(* IEC 61131-3 sources: teller/JD_Teller_LC2_V11/Class/Box_Editor_Preview_TC, 1 file *)

(* ---- Box_Editor_Preview_TC.st ---- *)
(*!
<Class
	Name               = "Box_Editor_Preview_TC"
	Revision           = "1.6"
	RealtimeTask       = "false"
	CyclicTask         = "false"
	BackgroundTask     = "false"
	Sigmatek           = "false"
	OSInterface        = "false"
	HighPriority       = "false"
	Automatic          = "false"
	UpdateMode         = "Prescan"
	SharedCommandTable = "true"
	Objectsize         = "(540,780)">
	<Channels>
		<Server Name="ClassSvr" Visualized="false" Initialize="false" WriteProtected="true" Retentive="false"/>
		<Server Name="s_Boxtype" Visualized="true" Initialize="false" WriteProtected="false" Retentive="false"/>
		<Server Name="s_Offset" Visualized="true" Initialize="false" WriteProtected="false" Retentive="false"/>
		<Server Name="s_Refresh" Visualized="false" Initialize="false" WriteProtected="false" Retentive="false"/>
		<Server Name="s_SaveTC" Visualized="false" Initialize="false" WriteProtected="false" Retentive="false"/>
		<Server Name="s_T" Visualized="true" Initialize="false" WriteProtected="false" Retentive="false"/>
		<Server Name="s_U" Visualized="true" Initialize="false" WriteProtected="false" Retentive="false"/>
		<Server Name="s_V" Visualized="true" Initialize="false" WriteProtected="false" Retentive="false"/>
		<Server Name="s_W" Visualized="true" Initialize="false" WriteProtected="false" Retentive="false"/>
		<Server Name="s_X" Visualized="true" Initialize="false" WriteProtected="false" Retentive="false"/>
		<Server Name="s_Y" Visualized="true" Initialize="false" WriteProtected="false" Retentive="false"/>
		<Server Name="s_Z" Visualized="true" Initialize="false" WriteProtected="false" Retentive="false"/>
		<Client Name="c_Comment_Read" Required="true" Internal="false"/>
		<Client Name="c_Comment_Write" Required="true" Internal="false"/>
		<Client Name="c_Doosdata" Required="true" Internal="false"/>
		<Client Name="c_ResetTellers" Required="false" Internal="false"/>
	</Channels>
	<RevDoku>
		<Owner Company="JD" Author="JVD"/>
		<Dokumentation Revision="1.6" Date="2014-01-27" Author="JVD" Company="JD" Description="commentaar verbeterd + tellers reset"/>
		<Dokumentation Revision="1.4" Date="2013-11-22" Author="JVD" Company="JD" Description="ResetLijm detectie teller"/>
		<Dokumentation Revision="1.3" Date="2013-09-21" Author="JVD" Company="JD" Description="input error opgelost"/>
		<Dokumentation Revision="1.1" Date="2012-10-11" Author="JVD" Company="JD" Description="&#13;&#10;"/>
		<Dokumentation Revision="1.0" Date="2012-01-12" Author="JVD" Company="JD" Description="-Het commentaar wat bij de boxeditor is ingevoerd wordt bij de preview weergegeven.&#13;&#10;-Het string classje Boxedit_command_preview dient te worden aangesloten"/>
	</RevDoku>
</Class>
*)
Box_Editor_Preview_TC : CLASS
  //Servers:
	ClassSvr 	: SvrChCmd_DINT;
	s_SaveTC 	: SvrCh_DINT;
	s_Refresh 	: SvrCh_DINT;
	s_Boxtype 	: SvrCh_DINT;
	s_T 	: SvrCh_DINT;
	s_U 	: SvrCh_DINT;
	s_V 	: SvrCh_DINT;
	s_W 	: SvrCh_DINT;
	s_X 	: SvrCh_DINT;
	s_Y 	: SvrCh_DINT;
	s_Z 	: SvrCh_DINT;
	s_Offset 	: SvrCh_DINT;
  //Clients:
	c_Doosdata 	: CltChCmd_RAMex;
	c_Comment_Read 	: CltChCmd_StringRAM;
	c_Comment_Write 	: CltChCmd_StringRAM;
	c_ResetTellers 	: CltCh_DINT;
  //Variables:
		Doosdata 	: ^tDoosParameters;
		data : ARRAY [0..49] OF USINT;

  //Functions:

	FUNCTION VIRTUAL GLOBAL Init;

	FUNCTION VIRTUAL GLOBAL s_SaveTC::Write
		VAR_INPUT
			input (EAX) 	: DINT;
		END_VAR
		VAR_OUTPUT
			result (EAX) 	: DINT;
		END_VAR;

	FUNCTION VIRTUAL GLOBAL s_Refresh::Write
		VAR_INPUT
			input (EAX) 	: DINT;
		END_VAR
		VAR_OUTPUT
			result (EAX) 	: DINT;
		END_VAR;
  //Tables:
	FUNCTION @STD
		VAR_OUTPUT
			ret_code	: CONFSTATES;
		END_VAR;
	FUNCTION GLOBAL TAB @CT_;
END_CLASS;

#pragma usingLtd RAMex
#pragma usingLtd StringRAM

FUNCTION VIRTUAL GLOBAL Box_Editor_Preview_TC::Init

  if c_DoosData.GetSize() <> sizeof(tDoosParameters) then
     c_DoosData.SetSize(udSize:=sizeof(tDoosParameters));
  end_if;

  if _FirstScan = 1 then
      DoosData := (c_DoosData.GetDataPtr())$^tDoosParameters;

      s_Boxtype  :=Doosdata^.Doostype;
      s_T := Doosdata^.T;
      s_U := Doosdata^.U;
      s_V := Doosdata^.V;
      s_W := Doosdata^.W;
      s_X := Doosdata^.X;
      s_Y := Doosdata^.Y;
      s_Z := Doosdata^.Z;
      s_Offset := Doosdata^.Offset;

  end_if;

END_FUNCTION

FUNCTION VIRTUAL GLOBAL Box_Editor_Preview_TC::s_SaveTC::Write
	VAR_INPUT
		input (EAX) 	: DINT;
	END_VAR
	VAR_OUTPUT
		result (EAX) 	: DINT;
	END_VAR

	s_SaveTC := input;
  s_SaveTC := 0;

  c_Comment_Write.Clear();
  _memset(dest:=#data[0], usByte:=0, cntr:=sizeof(data));

  if    c_Comment_Read.GetLength() > 0 then
        c_Comment_Read.ReadDataOff(udOff:=0, pData:=#data[0], udMax:=sizeof(data));
        c_Comment_Write.WriteDataOff(udLen:= c_Comment_Read.GetLength(), udOff:= 0, pData:=#data[0] );
  end_if;

  s_Boxtype  :=Doosdata^.Doostype;
  s_T := Doosdata^.T;
  s_U := Doosdata^.U;
  s_V := Doosdata^.V;
  s_W := Doosdata^.W;
  s_X := Doosdata^.X;
  s_Y := Doosdata^.Y;
  s_Z := Doosdata^.Z;
  s_Offset := Doosdata^.Offset;

 	result := s_SaveTC;

END_FUNCTION

FUNCTION VIRTUAL GLOBAL Box_Editor_Preview_TC::s_Refresh::Write
	VAR_INPUT
		input (EAX) 	: DINT;
	END_VAR
	VAR_OUTPUT
		result (EAX) 	: DINT;
	END_VAR

	s_Refresh := input;
  s_Refresh := 0;

  c_Comment_Write.Clear();
  _memset(dest:=#data[0], usByte:=0, cntr:=sizeof(data));

  if    c_Comment_Read.GetLength() > 0 then
        c_Comment_Read.ReadDataOff(udOff:=0, pData:=#data[0], udMax:=sizeof(data));
        c_Comment_Write.WriteDataOff(udLen:= c_Comment_Read.GetLength(), udOff:= 0, pData:=#data[0] );
  end_if;

  s_Boxtype  :=Doosdata^.Doostype;
  s_T := Doosdata^.T;
  s_U := Doosdata^.U;
  s_V := Doosdata^.V;
  s_W := Doosdata^.W;
  s_X := Doosdata^.X;
  s_Y := Doosdata^.Y;
  s_Z := Doosdata^.Z;
  s_Offset := Doosdata^.Offset;

  c_ResetTellers.Write(input:=1);

 	result := s_Refresh;

END_FUNCTION
